// TIA Portal V17 export
// export: Created 2024-06-16T17:47:39.4535187Z, ExportSetting WithDefaults, DisplayName Totally Integrated Automation Portal, DisplayVersion V17, DisplayName TIA Portal Openness, DisplayVersion V17, DisplayName TIA Portal Version Control Interface, DisplayVersion V17, DisplayName STEP 7 Professional, DisplayVersion V17, DisplayName STEP 7 Safety, DisplayVersion V17, DisplayName WinCC Professional, DisplayVersion V17
VAR_GLOBAL   // PLC tag table "St2_In"
   IO_Cpt_V1 AT %I2.1 : Bool;   // Présence barquette en début de Vision : V1
   IO_Cpt_V2 AT %I2.2 : Bool;   // Détection butée à came : V2
   IO_Cpt_V3 AT %I2.3 : Bool;   // Détection butée pivot : V3
END_VAR
